PROGRAM Q7
VAR
	button_up 	: BOOL 	:= FALSE;
	moving		: BOOL 	:= FALSE;
	
END_VAR

// When the up button is pressed, the moving status indicator will toggle

// To run this program, paste the following into MAIN, then interact with the Visualisation Q7_V
// Q7();
VAR // added by the converter: edge detectors and wires of the graphical bodies
    _w1 : BOOL;
END_VAR

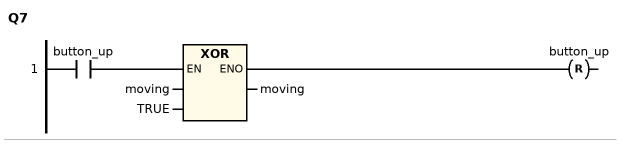
// NETWORK 1
_w1 := button_up;
IF _w1 THEN moving := moving XOR TRUE; END_IF
button_up R= _w1;

END_PROGRAM

(* stored: Version 1.1.0.1, ProductVersion 3.1.4024.12
   POU Q7: Id {25cd2fe7-3b40-4187-b4ac-dad177ff2fd5}, SpecialFunc None *)
